(* PLC project PLC107_DI, home PLC107_DI 1 *)
(* stored: creationDateTime 2019-11-13T09:37:45, productRelease 0, modificationDateTime 2020-07-16T10:10:52, version 1 *)

(* Установка режима работы дискретного входа *)
FUNCTION_BLOCK DIMode
  VAR_INPUT
    Ex : BOOL := FALSE;  (* разрешение на выполнение *)
    DIn : BYTE := 0;  (* номер входа *)
    M : BYTE := 0;  (* режим работы *)
  END_VAR
  VAR_OUTPUT
    Om : BYTE := 0;  (* режим работы (установленный) *)
    Ok : BYTE := 0;  (* код результата исполнения блока *)
  END_VAR

            {extern void App_DIMode(DIMODE*);App_DIMode(data__);}

          
END_FUNCTION_BLOCK

(* Получить значение нормального дискретного входа *)
FUNCTION_BLOCK DIVal
  VAR_INPUT
    Ex : BOOL := FALSE;  (* разрешение на выполнение *)
    DIn : BYTE := 0;  (* номер входа *)
  END_VAR
  VAR_OUTPUT
    Ov : BOOL := FALSE;  (* значение *)
    Ok : BYTE := 0;  (* код результата исполнения блока *)
  END_VAR

            {extern void App_DIVal(DIVAL*);App_DIVal(data__);}

          
END_FUNCTION_BLOCK

(* Получить значение входа тахометра *)
FUNCTION_BLOCK DICntT
  VAR_INPUT
    Ex : BOOL := FALSE;  (* разрешение на выполнение *)
    DIn : BYTE := 0;  (* номер входа *)
    Ref : WORD := 0;  (* уставка *)
    RefEn : BOOL := FALSE;  (* разрешение работы по уставке *)
  END_VAR
  VAR_OUTPUT
    Ov : WORD := 0;  (* значение *)
    Oref : BOOL := FALSE;  (* признак достижения уставки *)
    Ok : BYTE := 0;  (* код результата исполнения блока *)
  END_VAR

            {extern void App_DICntT(DICNTT*);App_DICntT(data__);}

          
END_FUNCTION_BLOCK

(* Получить значение счетного входа *)
FUNCTION_BLOCK DICnt
  VAR_INPUT
    Ex : BOOL := FALSE;  (* разрешение на выполнение *)
    DIn : BYTE := 0;  (* номер входа *)
    Ref : DWORD := 0;  (* уставка *)
    RefEn : BOOL := FALSE;  (* разрешение работы по уставке *)
  END_VAR
  VAR_OUTPUT
    Ov : DWORD := 0;  (* значение счетчика *)
    Oref : BOOL := FALSE;  (* признак достижения уставки *)
    Ok : BYTE := 0;  (* код результата исполнения блока *)
  END_VAR

            {extern void App_DICnt(DICNT*);App_DICnt(data__);}

          
END_FUNCTION_BLOCK

(* Сброс счетного входа или входа тахометра *)
FUNCTION_BLOCK DICntRst
  VAR_INPUT
    Ex : BOOL := FALSE;  (* разрешение на выполнение *)
    DIn : BYTE := 0;  (* номер входа *)
    Rst : BOOL := FALSE;  (* команда сброса *)
  END_VAR
  VAR_OUTPUT
    Ok : BYTE := 0;  (* код результата исполнения блока *)
  END_VAR

            {extern void App_DICntRst(DICNTRST*);App_DICntRst(data__);}

          
END_FUNCTION_BLOCK

(* Получить значения входов счетного энкодера *)
FUNCTION_BLOCK DIEnc
  VAR_INPUT
    Ex : BOOL := FALSE;  (* разрешение на выполнение *)
    DIn : BYTE := 0;  (* номер первичного группового входа *)
    RefA : DWORD := 0;  (* уставка счетчика фазы A *)
    RefAEn : BOOL := FALSE;  (* разрешение работы счетчика фазы A по уставке *)
    RefB : DWORD := 0;  (* уставка счетчика фазы B *)
    RefBEn : BOOL := FALSE;  (* разрешение работы счетчика фазы B по уставке *)
    RefT : WORD := 0;  (* уставка тахометра *)
    RefTEn : BOOL := FALSE;  (* разрешение работы тахометра по уставке *)
  END_VAR
  VAR_OUTPUT
    OA : DWORD := 0;  (* значение счетчика фазы A *)
    OAref : BOOL := FALSE;  (* признак достижения уставки счетчиком фазы A *)
    OB : DWORD := 0;  (* значение счетчика фазы B *)
    OBref : BOOL := FALSE;  (* признак достижения уставки счетчиком фазы B *)
    OT : WORD := 0;  (* значение тахометра *)
    OTref : BOOL := FALSE;  (* признак достижения уставки тахометром *)
    Ok : BYTE := 0;  (* код результата исполнения блока *)
  END_VAR

            {extern void App_DIEnc(DIENC*);App_DIEnc(data__);}

          
END_FUNCTION_BLOCK
